PROGRAM MAIN
VAR
	 E_STOP_ftring                                   :F_TRIG;
     E_STOP_rtring                                   :R_TRIG;
	 E_STOP_rem_rtring                         :R_TRIG;
     E_STOP_rem_ftring                         :F_TRIG;
	 Axis_All_Positionstart_rtrig				:R_TRIG;

END_VAR

UPSPersitent();
INIT();
Axis1_FC();
Axis2_FC();
IF simulation THEN
	E_STOP:=TRUE;
	foreward_limit_axis1:=TRUE;
	backward_limit_axis1:=TRUE;
	foreward_limit_axis2:=TRUE;
	backward_limit_axis2:=TRUE;
END_IF
// E_STOP_ftring(CLK:=E_STOP , Q=> );
Axis_All_Positionstart_rtrig(CLK:=Axis_All_Positionstart,Q=>);
IF Axis_All_Positionstart_rtrig. Q THEN
	Axis1_Positionstart:=TRUE;
	Axis2_Positionstart:=TRUE;
	//Axis_All_Positionstart:=FALSE;
END_IF
(*
IF Axis_All_PositiveJog THEN
	Axis1_PositiveJog:=TRUE;
	Axis2_PositiveJog:=TRUE;
	Axis_All_PositiveJog:=FALSE;
END_IF
IF Axis_All_NegativeJog THEN
	Axis1_NegativeJog:=TRUE;
	Axis1_NegativeJog:=TRUE;
	Axis_All_NegativeJog:=FALSE;
END_IF
*)
(*
IF Axis_All_STOP THEN
	Axis1_STOP:=TRUE;
	Axis2_STOP:=TRUE;
	Axis_All_STOP:=FALSE;
END_IF
*)
 
IF E_STOP  AND NOT Axis1_error AND NOT Axis2_error AND touchLimitSwitch_axis1 AND touchLimitSwitch_axis2 THEN
	Error:=FALSE;//无错误
ELSE
	Error:=TRUE;//无错误
END_IF
InputPositionProtection();
LVDT();
touchLimitSwitch_axis1:=foreward_limit_axis1 AND backward_limit_axis1;
touchLimitSwitch_axis2:=foreward_limit_axis2 AND backward_limit_axis2;
modbus();
(*******控制模式选择及显示，在电机运行过程中禁止切换*********)   
 IF  Local_Remote   THEN
      Local_led                       := TRUE;
      Remote_led                      := FALSE;  
   ELSE	
      Local_led                       := FALSE;
      Remote_led                      := TRUE;
 END_IF;


(***********急停************)
    E_STOP_ftring(CLK:=E_STOP , Q=> );
    E_STOP_rtring(CLK:=E_STOP , Q=> );
    E_STOP_rem_ftring(CLK:=E_STOP_rem , Q=> );
    E_STOP_rem_rtring(CLK:=E_STOP_rem , Q=> );
IF   E_STOP_rem   OR  NOT  E_STOP THEN     
     E_STOP_led      := TRUE;	
     power_do1                          := FALSE;     
     power_do2                          := FALSE;
     	 
END_IF;

//本地上升沿触发且远程FALSE；或者远程下降沿触发且本地急停TRUE
IF  (E_STOP_rtring.Q AND  NOT  E_STOP_rem) OR ( E_STOP AND E_STOP_rem_ftring.Q ) THEN
E_STOP_led     := FALSE;
END_IF;

(********实际温度值********)
TempController1_PV  :=35.0*( (INT_TO_REAL(PT1_IN))*10.0/32767)-50.0;//接入EL3214，三线制pt100
TempController2_PV  :=35.0*( (INT_TO_REAL(PT2_IN))*10.0/32767)-50.0;//接入EL3214，三线制pt100

END_PROGRAM

(* stored: Version 1.1.0.1, ProductVersion 3.1.4024.6
   POU MAIN: Id {ea8307cc-ac85-49ab-b5fb-1ec00128eeda}, SpecialFunc None *)
